Fanuc KAREL source: kt00401.KL

-- PROVISIONAL review KL for V940-1; original PC SHA256 192394c09ef31364ae1069c742604759fcfa1f86e8affec16ef9067e57585723
-- Incomplete behavior may be omitted. Consult companion uncertainty JSON. Do not deploy.
PROGRAM KT00401
%NOLOCKGROUP
VAR
  I1 : INTEGER
  I2 : INTEGER
  OUT : BOOLEAN
BEGIN
  -- V9_ZERO_TABLE_METADATA_HINT layout=0001; no indexed target words; source/name/runtime held
  -- UNRESOLVED_PC offsets 5-16; opcodes 2E,23
  -- UNRESOLVED_PC offsets 21-32; opcodes 2E,23
  -- UNRESOLVED_PC offsets 37-48; opcodes 2E,23
  -- UNRESOLVED_PC offsets 53-64; opcodes 2E,23
  -- UNRESOLVED_PC offsets 69-88; opcodes 21,21,5B,23
  -- UNRESOLVED_PC offsets 93-97; opcodes 7F
END KT00401
